// TIA Portal V17 export
// export: Created 2025-03-10T12:19:12.3105176Z, ExportSetting WithDefaults, DisplayName Totally Integrated Automation Portal, DisplayVersion V17 Update 8, DisplayName TIA Portal Openness, DisplayVersion V17 Update 8, DisplayName TIA Portal Version Control Interface, DisplayVersion V17, DisplayName SINAMICS Startdrive Advanced, DisplayVersion V17 SP2, DisplayName SINAMICS Startdrive G110M, G120, G120C, G120D, G120P, G115D, DisplayVersion V17 SP2, DisplayName SINAMICS Startdrive G130, G150, S120, S150, SINAMICS MV, S210, DisplayVersion V17 SP2, DisplayName STEP 7 Professional, DisplayVersion V17 Update 8, DisplayName SINUMERIK ONE STEP 7 Toolbox, DisplayVersion V17 Update 12, DisplayName SINUMERIK 840D sl STEP 7 Toolbox, DisplayVersion V17 Update 12, DisplayName STEP 7 Safety, DisplayVersion V17 Update 6, DisplayName WinCC Advanced, DisplayVersion V17 Update 8
DATA_BLOCK "DB22532_STIRRER_CONTROL_HOPPER_2_UNIT_02"   // DB22532
{ DB_Accessible_From_OPC_UA := 'FALSE' }
VERSION : 0.1
// stored: AutoNumber false, DBAccessibleFromOPCUA false, DBAccessibleFromWebserver true, InstanceOfName FB22502_STIRRER_CONTROL, InstanceOfType FB
"FB22502_STIRRER_CONTROL"
   // VAR_INPUT
   //    CONTROL_ON_DELAYED : Bool;
   //    MOTOR_CONDITIONS : Bool;
   //    MOTOR_STATUS_ERROR : Bool;
   //    MOTOR_STATUS_ENABLE : Bool;
   //    MOTOR_STATUS_REACHED : Bool;
   //    START_MANUAL_REQUEST : Bool;
   //    START_SEMI_REQUEST : Bool;
   //    START_AUTO_REQUEST : Bool;
   //    START_PROGRAM_REQUEST : Bool;
   //    STOP_MANUAL_REQUEST : Bool;
   //    STOP_SEMI_REQUEST : Bool;
   //    STOP_AUTO_REQUEST : Bool;
   //    STOP_PROGRAM_REQUEST : Bool;
   //    MOTOR_ACTUAL_POSITION : DInt;
   //    MOTOR_ACTUAL_VELOCITY : DInt;
   //    MOTOR_ACTUAL_CURRENT : DInt;
   //    MOTOR_ACTUAL_CURRENT_FILTERED : DInt;
   //    MOTOR_ACTUAL_TEMPERATURE : Real;
   //    MOTOR_STATUS_REGISTER : UDInt;
   // END_VAR
   // VAR_OUTPUT
   //    "MOTOR _VELOCITY _TARGET _SOURCE" : DInt;
   //    "MOTOR _MODE _OF _OPERATION" : Int;
   //    "MOTOR _ENABLE _POWER _STAGE" : Int;
   //    "MOTOR _OUT1" : Bool;
   //    "MOTOR _OUT2" : Bool;
   //    "MOTOR _OUT3" : Bool;
   //    "MOTOR _ENABLE _1" : Bool;
   //    "MOTOR _ENABLE _2" : Bool;
   //    "CURRENT _LIMIT _ALARM" : Bool;
   //    "TEMPRETATURE _LIMIT _ALARM" : Bool;
   // END_VAR
   // VAR
   //    DATA_STANDARD : "GENERAL_DATA_START_STOP";
   //    DATA_HMI : "HMI_DATA_START_STOP";
   //    INPUT_SETTINGS : Struct
   //       UNIT_NUMBER : Int := 2;
   //       HOPPER_NUMBER : Int := 2;
   //    END_STRUCT;
   //    ALARM_SETTINGS : Struct
   //       CURRENT_LIMIT : DInt;
   //       TEMPERATURE_LIMIT : Real;
   //       TIMER_CURRENT_LIMIT : TON_TIME;
   //       TIMER_TEMPERATURE_LIMIT : TON_TIME;
   //    END_STRUCT;
   //    "HMI _SETPOINT _VELOCITY" : DInt;
   //    "HMI _ACTUAL _POSITION" : DInt;
   //    "HMI _ACTUAL _VELOCITY" : DInt;
   //    "HMI _ACTUAL _CURRENT" : DInt;
   //    "HMI _ACTUAL _CURRENT _FILTERED" : DInt;
   //    "HMI _STIRRER _LOW _RANGE" : DInt;
   //    "HMI _STIRRER _HIGH _RANGE" : DInt;
   //    "PROGRAM _SETPOINT _VELOCITY" : DInt;
   //    "SETPOINT _VELOCITY" : DInt;
   //    "FEEDBACK _POSITION" : DInt;
   //    "FEEDBACK _VELOCITY" : DInt;
   //    "FEEDBACK _CURRENT" : DInt;
   //    "FEEDBACK _CURRENT _FILTERED" : DInt;
   //    "FEEDBACK _TEMPERATURE" : Real;
   // END_VAR
BEGIN
END_DATA_BLOCK
